// TIA Portal V18 export
// export: Created 2026-01-09T11:31:58.6798888Z, ExportSetting WithDefaults, DisplayName Totally Integrated Automation Portal, DisplayVersion V18 Update 5, DisplayName TIA Portal Openness, DisplayVersion V18 Update 5, DisplayName TIA Portal Teamcenter Gateway, DisplayVersion V18, DisplayName TIA Portal Version Control Interface, DisplayVersion V18, DisplayName SINAMICS Startdrive Advanced, DisplayVersion V18 SP2 Update 1, DisplayName SINAMICS Startdrive G110M, G120, G120C, G120D, G120P, G115D, DisplayVersion V18 SP2 Update 1, DisplayName SINAMICS Startdrive G130, G150, S120, S150, SINAMICS MV, S210, G220, S200, DisplayVersion V18 SP2 Update 1, DisplayName STEP 7 Professional, DisplayVersion V18 Update 5, DisplayName STEP 7 Safety, DisplayVersion V18, DisplayName WinCC Professional, DisplayVersion V18 Update 5
TagTable "DeviceErrorWord"
  A1TableScan : Word  (%DB1067.DBW100, CPU S71500-2PN_TP700, 500 ms)
  A1TableUnloading : Word  (%DB1067.DBW102, CPU S71500-2PN_TP700, 500 ms)
  A1RotaryScan : Word  (%DB1067.DBW104, CPU S71500-2PN_TP700, 500 ms)
  Robot_1 : Word  (%DB1067.DBW150, CPU S71500-2PN_TP700, 500 ms)
  A1FixtureCodeScan : Word  (%DB1067.DBW106, CPU S71500-2PN_TP700, 500 ms)
  A2TableScan : Word  (%DB1067.DBW108, CPU S71500-2PN_TP700, 500 ms)
  A2TableUnloading : Word  (%DB1067.DBW110, CPU S71500-2PN_TP700, 500 ms)
  A2RotaryScan : Word  (%DB1067.DBW112, CPU S71500-2PN_TP700, 500 ms)
  B1Press : Word  (%DB1067.DBW120, CPU S71500-2PN_TP700, 500 ms)
  B2Press : Word  (%DB1067.DBW122, CPU S71500-2PN_TP700, 500 ms)
  CGlueing : Word  (%DB1067.DBW130, CPU S71500-2PN_TP700, 500 ms)
  NG_1 : Word  (%DB1067.DBW140, CPU S71500-2PN_TP700, 500 ms)
  Robot_2 : Word  (%DB1067.DBW152, CPU S71500-2PN_TP700, 500 ms)
  Robot_3 : Word  (%DB1067.DBW154, CPU S71500-2PN_TP700, 500 ms)
  A2FixtureCodeScan : Word  (%DB1067.DBW114, CPU S71500-2PN_TP700, 500 ms)
  NG_2 : Word  (%DB1067.DBW142, CPU S71500-2PN_TP700, 500 ms)
  ShaftLine : Word  (%DB1067.DBW160, CPU S71500-2PN_TP700, 500 ms)
  MagnetLine : Word  (%DB1067.DBW170, CPU S71500-2PN_TP700, 500 ms)
  ReserveLine : Word  (%DB1067.DBW180, CPU S71500-2PN_TP700, 500 ms)
  UnloadingLine : Word  (%DB1067.DBW190, CPU S71500-2PN_TP700, 500 ms)
  CuringOven : Word  (%DB1067.DBW192, CPU S71500-2PN_TP700, 500 ms)
  A_Other : Word  (%DB1067.DBW116, CPU S71500-2PN_TP700, 1 s)
  C_Other : Word  (%DB1067.DBW142, CPU S71500-2PN_TP700, 1 s)
  MESS_Error : Word  (%DB1067.DBW200, CPU S71500-2PN_TP700, 1 s)
  A_DeviceError : Word  (%DB1067.DBW118, CPU S71500-2PN_TP700, 1 s)
  B_DeviceError : Word  (%DB1067.DBW124, CPU S71500-2PN_TP700, 1 s)
  C_DeviceError : Word  (%DB1067.DBW134, CPU S71500-2PN_TP700, 1 s)
  E_DeviceError : Word  (%DB1067.DBW144, CPU S71500-2PN_TP700, 1 s)
  F_DeviceError : Word  (%DB1067.DBW156, CPU S71500-2PN_TP700, 1 s)
  H_DeviceError : Word  (%DB1067.DBW162, CPU S71500-2PN_TP700, 1 s)
  J_DeviceError : Word  (%DB1067.DBW172, CPU S71500-2PN_TP700, 1 s)
  K_DeviceError : Word  (%DB1067.DBW182, CPU S71500-2PN_TP700, 1 s)
  L_DeviceError : Word  (%DB1067.DBW194, CPU S71500-2PN_TP700, 1 s)
